Staubli VAL3: enableLatch.pgx

program enableLatch()
begin
  // This program enable the Latch functionnality of the
  // WAGO750-631 module
  if (diEncLatched==false)
    doEnableLatch=true
  endIf
end
